(* IEC 61131-3 sources: volt/packages/volt-lsp-iec/test-corpus/lenze-mid/Device/Plc Logic/Application/Library Manager/RecipeManagement, 99 files *)

(* ---- IEC_ANYTYPE.dut ---- *)
TYPE IEC_ANYTYPE :
STRUCT
	PDATA : POINTER TO BYTE;
	TYPEOF : IEC_DataType;
	SIZE : UINT;
END_STRUCT
END_TYPE

(* ---- IEC_DATATYPE.dut ---- *)
TYPE IEC_DATATYPE :
(
	TYPE_BOOL,
	TYPE_INT,
	TYPE_BYTE,
	TYPE_WORD,
	TYPE_DINT,
	TYPE_DWORD,
	TYPE_REAL,
	TYPE_TIME,
	TYPE_STRING,
	TYPE_SINT,
	TYPE_USINT,
	TYPE_UINT,
	TYPE_UDINT,
	TYPE_DATE,
	TYPE_TOD,
	TYPE_DT,
	TYPE_LREAL,
	TYPE_LINT,
	TYPE_ULINT,
	TYPE_LWORD,
	TYPE_NONE,
	TYPE_BIT,
	TYPE_WSTRING,
	TYPE_LDATE,
	TYPE_LTOD,
	TYPE_LDT,
	TYPE_LTIME,
	TYPE_MAXTYPES
);
END_TYPE

(* ---- INFOVALUES.dut ---- *)
TYPE INFOVALUES :
(
	NO_INFO := 16#0,
	INFO_RECIPE_MANAGER_NOT_ALL_VARIABLES_FOUND := 16#1,
	INFO_RECIPE_MANAGER_OTHER_VARIABLES_FOUND := 16#2,
	INFO_RECIPE_MANAGER_ONE_OR_MORE_VARIABLES_FOUND := 16#4,
	INFO_RECIPE_MANAGER_ALL_VARIABLES_FOUND := 16#8
);
END_TYPE

(* ---- MEMBERSTOREDUCESTACKSIZE.dut ---- *)
TYPE MEMBERSTOREDUCESTACKSIZE :
STRUCT
	STFILE : STRING(512);
	TOKENIZER : RecipeManTokenizer;
	STPATHSEPARATOR : STRING(2);
	STHELP : STRING(512);
	STHELPPREVDIR : STRING(512);
	STCURRENTDIR : STRING(512);
	STLINEHELP : STRING(256);
	WSTVALUE : WSTRING(128);
	STHELPVALUE : STRING(256);
	STNAME : STRING(256);
	STRHELP : STRING(256);
END_STRUCT
END_TYPE

(* ---- MESSAGEBOX_STRUCT.dut ---- *)
TYPE MESSAGEBOX_STRUCT :
STRUCT
	EMESSAGEBOXDIALOGTYPES : DWORD;
	STITLE : STRING;
	SMESSAGETXT : STRING(1024);
END_STRUCT
END_TYPE

(* ---- PERSISTANTLOADTYPE.dut ---- *)
TYPE PERSISTANTLOADTYPE :
(
	LOAD_TYPE_NONE,
	LOAD_TYPE_SEARCH_FOR_NAME,
	LOAD_TYPE_SEARCH_FOR_VARNAME,
	LOAD_MATCHING_VARIABLES_BY_VARIABLENAME
);
END_TYPE

(* ---- RECIPEDATA.dut ---- *)
TYPE RECIPEDATA :
STRUCT
	PDATA : POINTER TO ARRAY [0..100000] OF RecipeDataValue;
	IDATACOUNT : DINT;
END_STRUCT
END_TYPE

(* ---- RECIPEDATAVALUE.dut ---- *)
TYPE RECIPEDATAVALUE :
STRUCT
	VALUE : IEC_AnyType;
END_STRUCT
END_TYPE

(* ---- RECIPEDESCRIPTION.dut ---- *)
TYPE RECIPEDESCRIPTION :
STRUCT
	STNAME : STRING;
	DATA : RecipeData;
	DESCDATA : RecipeDescriptionData;
END_STRUCT
END_TYPE

(* ---- RECIPEDESCRIPTIONDATA.dut ---- *)
TYPE RECIPEDESCRIPTIONDATA :
STRUCT
	PDATA : POINTER TO ARRAY [0..100000] OF RecipeVariableDescription;
	ICOUNT : DINT;
END_STRUCT
END_TYPE

(* ---- RECIPEMANENUMCOLUMNS.dut ---- *)
TYPE RECIPEMANENUMCOLUMNS :
(
	C_VARNAME,
	C_VALUE,
	C_TYPE,
	C_NAME,
	C_COMMENT,
	C_MIN,
	C_MAX
);
END_TYPE

(* ---- RECIPEREMOTEVARIABLE.dut ---- *)
TYPE RECIPEREMOTEVARIABLE :
STRUCT
	PBTINSTANCEPATH : POINTER TO BYTE;
END_STRUCT
END_TYPE

(* ---- RECIPEREMOTEVARIABLES.dut ---- *)
TYPE RECIPEREMOTEVARIABLES :
STRUCT
	PVARIABLES : POINTER TO RecipeRemoteVariable;
	DICOUNT : DINT;
END_STRUCT
END_TYPE

(* ---- RECIPESTORE.dut ---- *)
TYPE RECIPESTORE :
STRUCT
	_STPATH : STRING(512) := '';
	_BAUTOSAVE : BOOL := TRUE;
END_STRUCT
END_TYPE

(* ---- RECIPEVARIABLEDESCRIPTION.dut ---- *)
TYPE RECIPEVARIABLEDESCRIPTION :
STRUCT
	PSTNAME : POINTER TO BYTE;
	TYPEOF : IEC_DataType;
	MINVALUE : IEC_AnyType;
	MAXVALUE : IEC_AnyType;
	PSTVARNAME : POINTER TO BYTE;
	PSTCOMMENT : POINTER TO BYTE;
	DWFLAGS : DWORD;
END_STRUCT
END_TYPE

(* ---- STRINGINTPAIR.dut ---- *)
TYPE STRINGINTPAIR :
STRUCT
	STVAL : STRING(40);
	IVAL : INT;
END_STRUCT
END_TYPE

(* ---- GVL_RECIPECONSTANTS.gvl ---- *)
VAR_GLOBAL
	INVALID_DEFINITION_INDEX : INT := -1;
	CANNOT_ADD_RECIPE : INT := -1;
	INVALID_RECIPE_INDEX : INT := -1;
	RECIPESTORE_STRLEN : INT := 40;
	OUTPUT_INFO : INT := 16#1;
	OUTPUT_WARNING : INT := 16#2;
	OUTPUT_ERROR : INT := 16#4;
	OUTPUT_DEBUG : INT := 16#10;
	ASCII_PIPE : BYTE := 16#7C;
	NULL : POINTER TO BYTE := 0;
END_VAR

(* ---- GVL_RECIPEMANAGEMENT_INTERN.gvl ---- *)
VAR_GLOBAL
	G_RECIPEMANAGERCOMPONENT : STRING := 'RecipeManager';
	G_RECIPEMANAGERHELP : IRecipeManager;
	G_RECIPEMANCOMMANDSHELP : POINTER TO RecipeManCommands;
END_VAR

(* ---- GVL_RECIPEMANAGEMENT_TEMP.gvl ---- *)
VAR_GLOBAL
END_VAR

(* ---- GVL_RECIPEMANCOMMANDS_INTERN.gvl ---- *)
VAR_GLOBAL
	G_SEM : RecipeSem;
	G_BRECIPEMANAGERLOCKED : BOOL := TRUE;
	G_STFILENAME : STRING(512);
END_VAR

(* ---- INTERFACEIDS.gvl ---- *)
VAR_GLOBAL
	ITFID_IGENERIC : DWORD := 0;
	ITFID_IRECIPEMANAGER : DWORD := 1;
	ITFID_IGENERALCOMMAND : DWORD := 2;
END_VAR

(* ---- RETURNVALUES.gvl ---- *)
VAR_GLOBAL
	ERR_OK : UDINT := 16#0;
	ERR_FAILED : UDINT := 16#1;
	ERR_PARAMETER : UDINT := 16#2;
	ERR_NOTINITIALIZED : UDINT := 16#3;
	ERR_NOTIMPLEMENTED : UDINT := 16#C;
	ERR_NO_OBJECT : UDINT := 16#10;
	ERR_NOMEMORY : UDINT := 16#11;
	ERR_RECIPE_FILE_NOT_FOUND : UDINT := 16#4000;
	ERR_RECIPE_MISMATCH : UDINT := 16#4001;
	ERR_RECIPE_SAVE_ERR : UDINT := 16#4002;
	ERR_RECIPE_NOT_FOUND : UDINT := 16#4003;
	ERR_RECIPE_DEFINITION_NOT_FOUND : UDINT := 16#4004;
	ERR_RECIPE_ALREADY_EXIST : UDINT := 16#4005;
	ERR_NO_RECIPE_MANAGER_SET : UDINT := 16#4006;
	ERR_RECIPE_NOT_ALL_VARIABLES_WERE_LOADED : UDINT := 16#4007;
	ERR_RECIPE_NOMEMORY : UDINT := 16#4008;
	ERR_RECIPE_MANAGER_LOCKED_DURING_ONLINE_CHANGE : UDINT := 16#4009;
	ERR_SOURCE_EXHAUSTED : UDINT := 16#40A0;
	ERR_TARGET_EXHAUSTED : UDINT := 16#40A1;
	ERR_SOURCE_ILLEGAL : UDINT := 16#40A2;
END_VAR

(* ---- VERSIONINFO.gvl ---- *)
VAR_GLOBAL
	RECIPEMANAGER_VERSION_ATLEAST_3_2_0_0 : INT := 0;
	RECIPEMANAGER_VERSION_ATLEAST_3_2_0_1 : INT := 0;
	RECIPEMANAGER_VERSION_ATLEAST_3_2_0_2 : INT := 0;
	RECIPEMANAGER_VERSION_ATLEAST_3_3_0_0 : INT := 0;
	RECIPEMANAGER_VERSION_ATLEAST_3_3_0_10 : INT := 0;
	RECIPEMANAGER_VERSION_ATLEAST_3_3_0_20 : INT := 0;
	RECIPEMANAGER_VERSION_ATLEAST_3_5_5 : INT := 0;
	RECIPEMANAGER_VERSION_ATLEAST_3_5_9 : INT := 0;
	RECIPEMANAGER_VERSION_ATLEAST_3_5_10 : INT := 0;
	RECIPEMANAGER_VERSION_ATLEAST_3_5_14 : INT := 0;
END_VAR

(* ---- IGENERIC.itf ---- *)
INTERFACE IGENERIC
END_INTERFACE

METHOD GETINTERFACE : POINTER TO BYTE
VAR_INPUT
	DWITFID : DWORD;
END_VAR
END_METHOD

(* ---- IPERSISTANTRECIPELIST.itf ---- *)
INTERFACE IPERSISTANTRECIPELIST
END_INTERFACE

METHOD FREERECIPE : BOOL
VAR_INPUT
	RECIPE : IRecipe;
END_VAR
END_METHOD

METHOD GETRECIPENAME : STRING
VAR_INPUT
	IINDEX : INT;
END_VAR
END_METHOD

METHOD GETRECIPENAMES : DWORD
VAR_INPUT
	PSTRINGS : POINTER TO ARRAY [0..0] OF STRING;
	ISIZE : INT;
	ISTARTINDEX : INT;
END_VAR
END_METHOD

METHOD RELOAD : DWORD
END_METHOD

(* ---- IPERSISTANTRECIPELISTSUPPORTSADD.itf ---- *)
INTERFACE IPERSISTANTRECIPELISTSUPPORTSADD
END_INTERFACE

METHOD ADDRECIPE : BOOL
VAR_INPUT
	STNAME : REFERENCE TO STRING;
END_VAR
END_METHOD

(* ---- IPERSISTENTRECIPEHELPER.itf ---- *)
INTERFACE IPERSISTENTRECIPEHELPER
END_INTERFACE

METHOD DELETERECIPE : BOOL
VAR_INPUT
	STNAME : STRING;
END_VAR
END_METHOD

METHOD GETFILEEXTENSION : STRING
END_METHOD

METHOD GETFILEPATH : STRING(512)
END_METHOD

METHOD LOADRECIPE : BOOL
VAR_INPUT
	DESC : REFERENCE TO RecipeDescription;
END_VAR
END_METHOD

METHOD LOADRECIPEFROM : BOOL
VAR_INPUT
	DESC : REFERENCE TO RecipeDescription;
	STFILE : REFERENCE TO STRING(255);
END_VAR
END_METHOD

METHOD SAVERECIPE : BOOL
VAR_INPUT
	DESC : REFERENCE TO RecipeDescription;
END_VAR
END_METHOD

METHOD SAVERECIPEAS : BOOL
VAR_INPUT
	DESC : REFERENCE TO RecipeDescription;
	STFILE : REFERENCE TO STRING(255);
END_VAR
END_METHOD

METHOD SETFILEPATH : BOOL
VAR_INPUT
	STPATH : STRING(512);
END_VAR
END_METHOD

(* ---- IRECIPE.itf ---- *)
INTERFACE IRECIPE
END_INTERFACE

METHOD FILLDESCRIPTION : BOOL
VAR_INPUT
	DESC : REFERENCE TO RecipeDescription;
END_VAR
END_METHOD

METHOD READ : BOOL
END_METHOD

METHOD UPDATEFROMDESCRIPTION : BOOL
VAR_INPUT
	DESC : REFERENCE TO RecipeDescription;
END_VAR
END_METHOD

METHOD WRITE : BOOL
END_METHOD

(* ---- IRECIPECHECKONSTART.itf ---- *)
INTERFACE IRECIPECHECKONSTART
END_INTERFACE

METHOD ALREADYEXISTING : BOOL
VAR_INPUT
	STNAME : STRING;
END_VAR
END_METHOD

METHOD GETALREADYEXISTINGRECIPES : BOOL
END_METHOD

(* ---- IRECIPEDEFINITION.itf ---- *)
INTERFACE IRECIPEDEFINITION
END_INTERFACE

METHOD CREATERECIPE : BOOL
VAR_INPUT
	STNAME : STRING;
	BREADCURRENT : BOOL;
	BSAVE : BOOL;
END_VAR
END_METHOD

METHOD FREERECIPE : BOOL
VAR_INPUT
	RECIPE : IRecipe;
END_VAR
END_METHOD

METHOD GETPERSISTENCYHELPER : POINTER TO IPersistentRecipeHelper
END_METHOD

METHOD GETRECIPE : RecipeDescription
VAR_INPUT
	IINDEX : INT;
END_VAR
END_METHOD

METHOD GETRECIPEINDEXBYNAME : INT
VAR_INPUT
	STNAME : STRING;
END_VAR
END_METHOD

METHOD GETRECIPENAME : STRING
VAR_INPUT
	IINDEX : INT;
END_VAR
END_METHOD

METHOD GETRECIPENAMES : DWORD
VAR_INPUT
	PSTRINGS : POINTER TO ARRAY [0..0] OF STRING;
	ISIZE : INT;
	ISTARTINDEX : INT;
END_VAR
END_METHOD

METHOD GETRECIPEVALUES : DWORD
VAR_INPUT
	PSTRINGS : POINTER TO ARRAY [0..0] OF STRING;
	ISIZE : INT;
	ISTARTINDEX : INT;
	ISTRINGLENGTH : INT;
END_VAR
END_METHOD

METHOD GETRECIPEVARIABLENAMES : DWORD
VAR_INPUT
	PSTRINGS : POINTER TO ARRAY [0..0] OF STRING;
	ISIZE : INT;
	ISTARTINDEX : INT;
END_VAR
END_METHOD

METHOD LOADALL : BOOL
VAR_INPUT
	BCLEAR : BOOL;
END_VAR
END_METHOD

METHOD REGISTEREVENTHANDLER : BOOL
VAR_INPUT
	HANDLER : IRecipeDefinitionEventHandler;
END_VAR
END_METHOD

METHOD RELOAD : DWORD
END_METHOD

METHOD SAVEALL : BOOL
END_METHOD

METHOD SELECTRECIPE : BOOL
VAR_INPUT
	IINDEX : INT;
END_VAR
END_METHOD

METHOD SETRECIPEVALUES : DWORD
VAR_INPUT
	PSTRINGS : POINTER TO ARRAY [0..0] OF STRING;
	ISIZE : INT;
	ISTARTINDEX : INT;
END_VAR
END_METHOD

METHOD UNREGISTEREVENTHANDLER : BOOL
VAR_INPUT
	HANDLER : IRecipeDefinitionEventHandler;
END_VAR
END_METHOD

(* ---- IRECIPEDEFINITION2.itf ---- *)
INTERFACE IRECIPEDEFINITION2
END_INTERFACE

METHOD GETRECIPEVARIABLECOUNT : DINT
END_METHOD

METHOD GETRECIPEVARIABLENAME : POINTER TO BYTE
VAR_INPUT
	IVARINDEX : DINT;
END_VAR
VAR_OUTPUT
	ERRORCODE : DWORD;
END_VAR
END_METHOD

(* ---- IRECIPEDEFINITION3.itf ---- *)
INTERFACE IRECIPEDEFINITION3
END_INTERFACE

METHOD GETRECIPEVALUESSIZEOF : DWORD
VAR_INPUT
	PSTRINGS : POINTER TO ARRAY [0..0] OF STRING;
	ISIZE : INT;
	ISTARTINDEX : INT;
	ISIZEOFSTRING : INT;
END_VAR
END_METHOD

(* ---- IRECIPEDEFINITIONEVENTHANDLER.itf ---- *)
INTERFACE IRECIPEDEFINITIONEVENTHANDLER
END_INTERFACE

METHOD AFTERCREATE : BOOL
END_METHOD

METHOD BEFORECLEAR : BOOL
END_METHOD

METHOD SELECTIONCHANGED : BOOL
END_METHOD

(* ---- IRECIPEFACTORY.itf ---- *)
INTERFACE IRECIPEFACTORY
END_INTERFACE

METHOD CREATERECIPE : IRecipe
VAR_INPUT
	STDEFINITIONNAME : STRING;
	STRECIPENAME : STRING;
END_VAR
END_METHOD

METHOD FREERECIPE : BOOL
VAR_INPUT
	STDEFINITIONNAME : STRING;
	REC : IRecipe;
END_VAR
END_METHOD

(* ---- IRECIPEMANAGER.itf ---- *)
INTERFACE IRECIPEMANAGER
END_INTERFACE

METHOD GETRECIPEDEFINITION : IRecipeDefinition
VAR_INPUT
	IINDEX : INT;
END_VAR
END_METHOD

METHOD GETRECIPEDEFINITIONBYNAME : IRecipeDefinition
VAR_INPUT
	STDEFINITIONNAME : STRING;
END_VAR
END_METHOD

METHOD GETRECIPEDEFINITIONINDEXBYNAME : INT
VAR_INPUT
	STDEFINITIONNAME : STRING;
END_VAR
END_METHOD

METHOD SELECTRECIPEDEFINITION : BOOL
VAR_INPUT
	IINDEX : INT;
END_VAR
END_METHOD

(* ---- IRECIPESELECTION.itf ---- *)
INTERFACE IRECIPESELECTION
END_INTERFACE

METHOD DELETE : BOOL
END_METHOD

METHOD LOAD : BOOL
END_METHOD

METHOD LOADFROM : BOOL
VAR_INPUT
	STNAME : REFERENCE TO STRING(255);
END_VAR
END_METHOD

METHOD READ : BOOL
END_METHOD

METHOD READNOSAVE : BOOL
END_METHOD

METHOD RELEASE : BOOL
END_METHOD

METHOD SAVE : BOOL
END_METHOD

METHOD SAVEAS : BOOL
VAR_INPUT
	STNAME : REFERENCE TO STRING(255);
END_VAR
END_METHOD

METHOD UPDATEFROMVALUES : BOOL
VAR_INPUT
	DESC : RecipeDescription;
END_VAR
END_METHOD

METHOD WRITE : BOOL
END_METHOD

(* ---- IRECIPESELECTIONWITHCOMPARE.itf ---- *)
INTERFACE IRECIPESELECTIONWITHCOMPARE
END_INTERFACE

METHOD COMPARE : BOOL
END_METHOD

(* ---- IRECIPEWITHCOMPARE.itf ---- *)
INTERFACE IRECIPEWITHCOMPARE
END_INTERFACE

METHOD COMPARE : BOOL
END_METHOD

(* ---- ASSERT.pou ---- *)
FUNCTION ASSERT : BOOL
VAR_INPUT
	BVAL : BOOL;
	STMESSAGE : STRING;
END_VAR
END_FUNCTION

(* ---- DOFORFBSAVEASRECIPE.pou ---- *)
FUNCTION DOFORFBSAVEASRECIPE : BOOL
VAR_INPUT
	MEMORYFORFBSAVEASRECIPE : POINTER TO BYTE;
	RECIPEMAN : IRecipeManager;
	COMMANDMANAGER : ICommandManager2;
	ICMD : INT;
END_VAR
END_FUNCTION

(* ---- PSTRCAT.pou ---- *)
FUNCTION PSTRCAT : DINT
VAR_INPUT
	PSTDEST : POINTER TO STRING;
	PSTSRC : POINTER TO STRING;
	DIDESTSIZE : DINT;
END_VAR
END_FUNCTION

(* ---- PSTRLEN.pou ---- *)
FUNCTION PSTRLEN : DINT
VAR_INPUT
	PSTRING : POINTER TO STRING;
END_VAR
END_FUNCTION

(* ---- PSTRNCPY.pou ---- *)
FUNCTION PSTRNCPY : DINT
VAR_INPUT
	PSTDEST : POINTER TO BYTE;
	PSTSRC : POINTER TO BYTE;
	DIDESTSIZE : DINT;
END_VAR
END_FUNCTION

(* ---- RECIPEDODATASOURCESEXCHANGE.pou ---- *)
FUNCTION RECIPEDODATASOURCESEXCHANGE : UDINT
VAR_INPUT
	VARIABLES : RecipeRemoteVariables;
	BWRITING : BOOL;
	RECIPEMANAGER : IRecipeManager;
	DATASOURCESMGR : IDatasources.IDatasourcesMgr;
END_VAR
END_FUNCTION

(* ---- RECIPEDODATASOURCESEXCHANGE2.pou ---- *)
FUNCTION RECIPEDODATASOURCESEXCHANGE2 : UDINT
VAR_INPUT
	VARIABLES : RecipeRemoteVariables;
	RECIPEDEFNAME : STRING;
	BWRITING : BOOL;
	RECIPEMANAGER : IRecipeManager;
	DATASOURCESMGR : IDatasources.IDatasourcesMgr;
END_VAR
END_FUNCTION

(* ---- RECIPELOG.pou ---- *)
FUNCTION RECIPELOG : BOOL
VAR_INPUT
	DICLASS : DINT;
	DIERROR : DINT;
	DIINFO : DINT;
	STMESSAGE : STRING(255);
END_VAR
END_FUNCTION

(* ---- RECIPEMAN_FCTANYFROMSTRING.pou ---- *)
FUNCTION RECIPEMAN_FCTANYFROMSTRING : BOOL
VAR_INPUT
	STRSOURCE : POINTER TO STRING;
	PVARADR : POINTER TO BYTE;
	DWVARTYPE : IEC_DataType;
END_VAR
END_FUNCTION

(* ---- RECIPEMAN_FCTANYTOSTRING.pou ---- *)
FUNCTION RECIPEMAN_FCTANYTOSTRING : BOOL
VAR_INPUT
	STRRESULT : POINTER TO STRING;
	PVARADR : POINTER TO BYTE;
	DWVARTYPE : IEC_DataType;
END_VAR
END_FUNCTION

(* ---- RECIPEMAN_FCTDATATYPETOSTRING.pou ---- *)
FUNCTION RECIPEMAN_FCTDATATYPETOSTRING : BOOL
VAR_INPUT
	STRRESULT : POINTER TO STRING;
	DWVARTYPE : IEC_DataType;
END_VAR
END_FUNCTION

(* ---- RECIPEMAN_FCTGETDATAVALUE.pou ---- *)
FUNCTION RECIPEMAN_FCTGETDATAVALUE : POINTER TO BYTE
VAR_INPUT
	VALUE : IEC_AnyType;
	PSTR : POINTER TO BYTE;
	IBUFFERSIZE : INT;
	PILEN : POINTER TO INT;
END_VAR
END_FUNCTION

(* ---- RECIPEMAN_FCTLREALFROMSTRING.pou ---- *)
FUNCTION RECIPEMAN_FCTLREALFROMSTRING : BOOL
VAR_INPUT
	STRSOURCE : POINTER TO STRING;
	PVARADR : POINTER TO LREAL;
END_VAR
END_FUNCTION

(* ---- RECIPEMAN_FCTLREALTOSTRING.pou ---- *)
FUNCTION RECIPEMAN_FCTLREALTOSTRING : BOOL
VAR_INPUT
	STRRESULT : POINTER TO STRING;
	PVARADR : POINTER TO LREAL;
END_VAR
END_FUNCTION

(* ---- RECIPEMAN_FCTSETDATAVALUE.pou ---- *)
FUNCTION RECIPEMAN_FCTSETDATAVALUE : BOOL
VAR_INPUT
	DATA : POINTER TO BYTE;
	VALUE : IEC_AnyType;
END_VAR
END_FUNCTION

(* ---- RECIPEMAN_FCTSTRINGTODATATYPE.pou ---- *)
FUNCTION RECIPEMAN_FCTSTRINGTODATATYPE : BOOL
VAR_INPUT
	STRRESULT : POINTER TO STRING;
	DWVARTYPE : POINTER TO IEC_DataType;
END_VAR
END_FUNCTION

(* ---- RECIPEMAN_FCTTYPECLASSTODATATYPE.pou ---- *)
FUNCTION RECIPEMAN_FCTTYPECLASSTODATATYPE : IEC_DataType
VAR_INPUT
	TC : TypeClass;
END_VAR
END_FUNCTION

(* ---- RECIPEMAN_FILEEXISTS.pou ---- *)
FUNCTION RECIPEMAN_FILEEXISTS : BOOL
VAR_INPUT
	STFILENAME : REFERENCE TO STRING(255);
END_VAR
END_FUNCTION

(* ---- RECIPEMANCREATEDIRECTORY.pou ---- *)
FUNCTION RECIPEMANCREATEDIRECTORY : DWORD
VAR_INPUT
	PSTPATH : POINTER TO STRING(512);
	PMTRSS : POINTER TO MembersToReduceStackSize;
END_VAR
END_FUNCTION

(* ---- RECIPEMANMASKSTRING.pou ---- *)
FUNCTION RECIPEMANMASKSTRING : STRING(256)
VAR_INPUT
	PSTR : POINTER TO STRING(256);
	BWITHSEPARATOR : BOOL;
	CHSEPARATOR : BYTE;
	BFORUTF8 : BOOL;
END_VAR
END_FUNCTION

(* ---- RECIPEMANMASKWSTRING.pou ---- *)
FUNCTION RECIPEMANMASKWSTRING : BOOL
VAR_INPUT
	PBYTEIN : POINTER TO ARRAY [0..0] OF BYTE;
	PBYTEOUT : POINTER TO ARRAY [0..0] OF BYTE;
	IBUFFERSIZE : INT;
	BFORUTF8 : BOOL;
END_VAR
END_FUNCTION

(* ---- RECIPEMANUNMASKSTRING.pou ---- *)
FUNCTION RECIPEMANUNMASKSTRING : STRING(256)
VAR_INPUT
	PSTR : POINTER TO STRING(256);
	BWITHSEPARATOR : BOOL;
	CHSEPARATOR : BYTE;
	BFORUTF8 : BOOL;
END_VAR
END_FUNCTION

(* ---- RECIPEMANUNMASKWSTRING.pou ---- *)
FUNCTION RECIPEMANUNMASKWSTRING : BOOL
VAR_INPUT
	PSTR : POINTER TO STRING(256);
	BFORUTF8 : BOOL;
END_VAR
END_FUNCTION

(* ---- RECIPEMANWSTRINGTOSTRING.pou ---- *)
FUNCTION RECIPEMANWSTRINGTOSTRING : BOOL
VAR_INPUT
	PWSTRINGFROM : POINTER TO WSTRING;
	PSTRINGTO : POINTER TO STRING;
END_VAR
END_FUNCTION

(* ---- RECIPEPSTRNCPY.pou ---- *)
FUNCTION RECIPEPSTRNCPY : DINT
VAR_INPUT
	PSTDEST : POINTER TO BYTE;
	PSTSRC : POINTER TO BYTE;
	DIDESTSIZE : DINT;
END_VAR
END_FUNCTION

(* ---- RECIPESTRCMP.pou ---- *)
FUNCTION RECIPESTRCMP : INT
VAR_INPUT
	PST1 : POINTER TO STRING;
	PST2 : POINTER TO STRING;
	BENDSWITH : BOOL;
END_VAR
END_FUNCTION

(* ---- UTILGETFILESIZE.pou ---- *)
FUNCTION UTILGETFILESIZE : __XWORD
VAR_INPUT
	DWHANDLE : SysFile.RTS_IEC_HANDLE;
	STFILENAME : REFERENCE TO STRING(255);
	PULRESULT : POINTER TO UDINT;
END_VAR
END_FUNCTION

(* ---- VISU_FCTGETRECIPEDEFINITION.pou ---- *)
FUNCTION VISU_FCTGETRECIPEDEFINITION : DWORD
VAR_INPUT
	DWPARAM1 : __XWORD;
	DWPARAM2 : __XWORD;
	RECIPEMANAGER : IRecipeManager;
END_VAR
VAR_OUTPUT
	_RECIPEDEFINITION : IRecipeDefinition;
END_VAR
END_FUNCTION

(* ---- VISU_FCTGETRECIPEDEFINITION2.pou ---- *)
FUNCTION VISU_FCTGETRECIPEDEFINITION2 : DWORD
VAR_INPUT
	DWPARAM1 : __XWORD;
	DWPARAM2 : __XWORD;
	RECIPEMANAGER : IRecipeManager;
	BNOCURRENTRECIPEDEFINITION : BOOL;
END_VAR
VAR_OUTPUT
	_RECIPEDEFINITION : IRecipeDefinition;
END_VAR
END_FUNCTION

(* ---- VISU_FCTGETRECIPESELECTION.pou ---- *)
FUNCTION VISU_FCTGETRECIPESELECTION : DWORD
VAR_INPUT
	DWPARAM1 : __XWORD;
	DWPARAM2 : __XWORD;
	RECIPEMANAGER : IRecipeManager;
END_VAR
VAR_OUTPUT
	_RECIPEDEFINITION : IRecipeDefinition;
	_RECIPESELECTION : IRecipeSelection;
END_VAR
END_FUNCTION

(* ---- VISU_FCTGETRECIPESELECTION2.pou ---- *)
FUNCTION VISU_FCTGETRECIPESELECTION2 : DWORD
VAR_INPUT
	DWPARAM1 : __XWORD;
	DWPARAM2 : __XWORD;
	RECIPEMANAGER : IRecipeManager;
	BNOCURRENTRECIPESELECTION : BOOL;
END_VAR
VAR_OUTPUT
	_RECIPEDEFINITION : IRecipeDefinition;
	_RECIPESELECTION : IRecipeSelection;
END_VAR
END_FUNCTION

(* ---- ABSTRACTFILEPARAMSCOMMAND.pou ---- *)
FUNCTION_BLOCK ABSTRACTFILEPARAMSCOMMAND EXTENDS AbstractGeneralCommand
END_FUNCTION_BLOCK

METHOD EXECUTE : __XWORD
VAR_INPUT
	DWPARAM1 : __XWORD;
	DWPARAM2 : __XWORD;
END_VAR
END_METHOD

METHOD EXECUTEONFILEPARAMS : DWORD
VAR_INPUT
	STRECIPEDEF : STRING;
	STRECIPENAME : STRING;
	STFILE : STRING(255);
END_VAR
END_METHOD

(* ---- ABSTRACTGENERALCOMMAND.pou ---- *)
FUNCTION_BLOCK ABSTRACTGENERALCOMMAND
VAR
	_ITFGENERALCOMMAND : IGeneralCommand2 := THIS^;
	_RECIPEMANAGER : IRecipeManager;
	S_BASECOMMANDS : RecipeManCommands;
END_VAR
END_FUNCTION_BLOCK

METHOD EXECUTE : __XWORD
VAR_INPUT
	DWPARAM1 : __XWORD;
	DWPARAM2 : __XWORD;
END_VAR
END_METHOD

METHOD GETINTERFACE : POINTER TO BYTE
VAR_INPUT
	DWITFID : DWORD;
END_VAR
END_METHOD

METHOD SETRECIPEMANAGER
VAR_INPUT
	RECIPEMANAGER : IRecipeManager;
END_VAR
END_METHOD

(* ---- ABSTRACTRECIPEANDDEFINITIONNAMECOMMAND.pou ---- *)
FUNCTION_BLOCK ABSTRACTRECIPEANDDEFINITIONNAMECOMMAND EXTENDS AbstractGeneralCommand
END_FUNCTION_BLOCK

METHOD EXECUTE : __XWORD
VAR_INPUT
	DWPARAM1 : __XWORD;
	DWPARAM2 : __XWORD;
END_VAR
END_METHOD

METHOD EXECUTEONRECIPEDEFINITIONANDRECIPENAME : DWORD
VAR_INPUT
	STRECIPEDEFINITIONNAME : STRING;
	STRECIPENAME : STRING;
END_VAR
END_METHOD

(* ---- BINARYMANYFILESPERSISTANTRECIPEHELPER.pou ---- *)
FUNCTION_BLOCK BINARYMANYFILESPERSISTANTRECIPEHELPER
VAR
	_STDEFNAME : STRING;
	_STEXTENSION : STRING(16) := '.binrecipe';
	_STPATH : STRING(512) := '';
	_RECIPEMANAGER : IRecipeManager;
	_DATABUFFER : ARRAY [0..MAX_BUFFER_SIZE] OF BYTE;
	_CURRENTDATAPOSITION : INT;
	_MTRSS : MembersToReduceStackSize;
	MAX_BUFFER_SIZE : INT := 2000;
	RECIPEDEFINITIONNAME : STRING;
END_VAR
END_FUNCTION_BLOCK

METHOD DELETERECIPE : BOOL
VAR_INPUT
	STNAME : STRING;
END_VAR
END_METHOD

METHOD GETFILEEXTENSION : STRING
END_METHOD

METHOD GETFILEPATH : STRING(512)
END_METHOD

METHOD LOADRECIPE : BOOL
VAR_INPUT
	DESC : REFERENCE TO RecipeDescription;
END_VAR
END_METHOD

METHOD LOADRECIPEFROM : BOOL
VAR_INPUT
	DESC : REFERENCE TO RecipeDescription;
	STFILE : REFERENCE TO STRING(255);
END_VAR
END_METHOD

METHOD SAVERECIPE : BOOL
VAR_INPUT
	DESC : REFERENCE TO RecipeDescription;
END_VAR
END_METHOD

METHOD SAVERECIPEAS : BOOL
VAR_INPUT
	DESC : REFERENCE TO RecipeDescription;
	STFILE : REFERENCE TO STRING(255);
END_VAR
END_METHOD

METHOD SETFILEPATH : BOOL
VAR_INPUT
	STPATH : STRING(512);
END_VAR
END_METHOD

METHOD SETRECIPEMANAGER
VAR_INPUT
	RECIPEMANAGER : IRecipeManager;
END_VAR
END_METHOD

METHOD PRVINITFILENAME : BOOL
VAR_INPUT
	STRECIPE : STRING;
END_VAR
END_METHOD

METHOD PRVMEMCOPY : BOOL
VAR_INPUT
	PMEMDEST : POINTER TO BYTE;
	PMEMSOURCE : POINTER TO BYTE;
	ISIZE : INT;
END_VAR
END_METHOD

METHOD PRVREADDATAVALUE : BOOL
VAR_INPUT
	VALUE : IEC_AnyType;
	DWFILE : SysFile.RTS_IEC_HANDLE;
END_VAR
END_METHOD

METHOD PRVREADVALUE : BOOL
VAR_INPUT
	PDATA : POINTER TO BYTE;
	TYPEOF : IEC_DataType;
	VALUESIZE : UINT;
	DWFILE : SysFile.RTS_IEC_HANDLE;
END_VAR
END_METHOD

METHOD PRVSAVERECIPEBUFFERED : BOOL
VAR_INPUT
	DESC : REFERENCE TO RecipeDescription;
	DWHANDLE : SysFile.RTS_IEC_HANDLE;
END_VAR
END_METHOD

METHOD PRVSETLASTERROR : BOOL
VAR_INPUT
	DWERROR : DWORD;
END_VAR
END_METHOD

METHOD PRVWRITEDATAVALUE : BOOL
VAR_INPUT
	VALUE : IEC_AnyType;
	DWFILE : SysFile.RTS_IEC_HANDLE;
END_VAR
END_METHOD

METHOD PRVWRITEVALUE : BOOL
VAR_INPUT
	PDATA : POINTER TO BYTE;
	ISIZE : INT;
	TYPEOF : IEC_DataType;
	DWFILE : SysFile.RTS_IEC_HANDLE;
END_VAR
END_METHOD

METHOD PRVWRITEVALUEBUFFERED : BOOL
VAR_INPUT
	DWFILE : SysFile.RTS_IEC_HANDLE;
	PDATA : POINTER TO BYTE;
	ISIZE : INT;
END_VAR
END_METHOD

(* ---- PERSISTANTRECIPELIST.pou ---- *)
FUNCTION_BLOCK PERSISTANTRECIPELIST
VAR_INPUT
	_IPERSISTENTRECIPEHELPER : IPersistentRecipeHelper;
END_VAR
VAR
	_RECIPESVECTOR : Collections.StringVector;
	_TOKENIZER : RecipeManTokenizer;
	_STATICMEM : ARRAY [0..(STATIC_RECIPE_NAMES_SIZE / 4)] OF DWORD;
	STATIC_RECIPE_NAMES_SIZE : DWORD := 2000;
	RECIPECOUNT : INT;
END_VAR
END_FUNCTION_BLOCK

METHOD ADDRECIPE : BOOL
VAR_INPUT
	STNAME : REFERENCE TO STRING;
END_VAR
END_METHOD

METHOD FB_EXIT : BOOL
VAR_INPUT
	BINCOPYCODE : BOOL;
END_VAR
END_METHOD

METHOD FB_INIT : BOOL
VAR_INPUT
	BINITRETAINS : BOOL;
	BINCOPYCODE : BOOL;
END_VAR
END_METHOD

METHOD FREERECIPE : BOOL
VAR_INPUT
	RECIPE : IRecipe;
END_VAR
END_METHOD

METHOD GETRECIPENAME : STRING
VAR_INPUT
	IINDEX : INT;
END_VAR
END_METHOD

METHOD GETRECIPENAMES : DWORD
VAR_INPUT
	PSTRINGS : POINTER TO ARRAY [0..0] OF STRING;
	ISIZE : INT;
	ISTARTINDEX : INT;
END_VAR
END_METHOD

METHOD RELOAD : DWORD
END_METHOD

METHOD PRVADD : BOOL
VAR_INPUT
	STRECIPEFILE : REFERENCE TO STRING;
END_VAR
END_METHOD

METHOD PRVCLEAR : BOOL
END_METHOD

(* ---- RECIPECOLLECTION.pou ---- *)
FUNCTION_BLOCK RECIPECOLLECTION
VAR
	_ASTATICRECIPES : ARRAY [0..STATIC_RECIPE_COUNT] OF IRecipe;
	_IUSEDRECIPES : INT;
	_PADYNAMICRECIPES : POINTER TO ARRAY [0..20] OF IRecipe := 0;
	_IDYNAMICALLOCCOUNT : INT;
	STATIC_RECIPE_COUNT : INT := 20;
	FIRST_DYNAMIC_ALLOC_COUNT : INT := 20;
	COUNT : INT;
END_VAR
END_FUNCTION_BLOCK

METHOD ADDRECIPE : BOOL
VAR_INPUT
	RECIPE : IRecipe;
END_VAR
END_METHOD

METHOD FB_EXIT : BOOL
VAR_INPUT
	BINCOPYCODE : BOOL;
END_VAR
END_METHOD

METHOD GETRECIPE : IRecipe
VAR_INPUT
	IINDEX : INT;
END_VAR
END_METHOD

METHOD GETRECIPENAMES : DWORD
VAR_INPUT
	PSTRINGS : POINTER TO ARRAY [0..0] OF STRING;
	ISIZE : INT;
	ISTARTINDEX : INT;
END_VAR
END_METHOD

METHOD REMOVERECIPE : BOOL
VAR_INPUT
	IINDEX : INT;
END_VAR
END_METHOD

(* ---- RECIPEDEFINITION.pou ---- *)
FUNCTION_BLOCK RECIPEDEFINITION
VAR
	_STNAME : STRING;
	_PERSISTANTRECIPELIST : PersistantRecipeList;
	_IRECIPELIST : IPersistantRecipeList;
	_ICURRENTRECIPE : IRecipe := 0;
	_RECIPECOLL : RecipeCollection;
	_EVENTHELPER : RecipeDefinitionEventHelper;
	_PPERSISTENCYHELPER : POINTER TO IPersistentRecipeHelper;
	_BAUTOSAVE : BOOL := TRUE;
	_RECDESC : RecipeDescription;
	_CURSOR : RecipeSelection;
	_ICURRENTINDEX : INT := -1;
	_IRETURNEDINDEX : INT := -1;
	_INTERNALRECDESC : RecipeDescription;
	_RECIPEMANAGER : IRecipeManager;
	_RECIPEFACTORY : IRecipeFactory;
	ARRALREADYEXISTINGFILES : POINTER TO ARRAY [0..0] OF STRING(80);
	_IALREADYEXISTINGRECIPES : INT;
	CURRENT : IRecipeSelection;
	CURRENTLYSELECTEDRECIPE : POINTER TO RecipeDescription;
	INTPERSISTENCY : BOOL;
	NAME : STRING;
	PRVCURRENTRECIPE : IRecipe;
	PRVRECIPELIST : IPersistantRecipeList;
	RECIPECOUNT : INT;
END_VAR
END_FUNCTION_BLOCK

METHOD ALREADYEXISTING : BOOL
VAR_INPUT
	STNAME : STRING;
END_VAR
END_METHOD

METHOD CREATERECIPE : BOOL
VAR_INPUT
	STNAME : STRING;
	BREADCURRENT : BOOL;
	BSAVE : BOOL;
END_VAR
END_METHOD

METHOD FB_EXIT : BOOL
VAR_INPUT
	BINCOPYCODE : BOOL;
END_VAR
END_METHOD

METHOD FREERECIPE : BOOL
VAR_INPUT
	RECIPE : IRecipe;
END_VAR
END_METHOD

METHOD GETALREADYEXISTINGRECIPES : BOOL
END_METHOD

METHOD GETPERSISTENCYHELPER : POINTER TO IPersistentRecipeHelper
END_METHOD

METHOD GETRECIPE : RecipeDescription
VAR_INPUT
	IINDEX : INT;
END_VAR
END_METHOD

METHOD GETRECIPEBYNAME : IRecipe
VAR_INPUT
	STNAME : REFERENCE TO STRING;
END_VAR
END_METHOD

METHOD GETRECIPEINDEXBYNAME : INT
VAR_INPUT
	STNAME : STRING;
END_VAR
END_METHOD

METHOD GETRECIPENAME : STRING
VAR_INPUT
	IINDEX : INT;
END_VAR
END_METHOD

METHOD GETRECIPENAMES : DWORD
VAR_INPUT
	PSTRINGS : POINTER TO ARRAY [0..0] OF STRING;
	ISIZE : INT;
	ISTARTINDEX : INT;
END_VAR
END_METHOD

METHOD GETRECIPEVALUES : DWORD
VAR_INPUT
	PSTRINGS : POINTER TO ARRAY [0..0] OF STRING;
	ISIZE : INT;
	ISTARTINDEX : INT;
	ISTRINGLENGTH : INT;
END_VAR
END_METHOD

METHOD GETRECIPEVALUESSIZEOF : DWORD
VAR_INPUT
	PSTRINGS : POINTER TO ARRAY [0..0] OF STRING;
	ISIZE : INT;
	ISTARTINDEX : INT;
	ISIZEOFSTRING : INT;
END_VAR
END_METHOD

METHOD GETRECIPEVARIABLECOUNT : DINT
END_METHOD

METHOD GETRECIPEVARIABLENAME : POINTER TO BYTE
VAR_INPUT
	IVARINDEX : DINT;
END_VAR
VAR_OUTPUT
	ERRORCODE : DWORD;
END_VAR
END_METHOD

METHOD GETRECIPEVARIABLENAMES : DWORD
VAR_INPUT
	PSTRINGS : POINTER TO ARRAY [0..0] OF STRING;
	ISIZE : INT;
	ISTARTINDEX : INT;
END_VAR
END_METHOD

METHOD LOADALL : BOOL
VAR_INPUT
	BCLEAR : BOOL;
END_VAR
END_METHOD

METHOD REGISTEREVENTHANDLER : BOOL
VAR_INPUT
	HANDLER : IRecipeDefinitionEventHandler;
END_VAR
END_METHOD

METHOD RELOAD : DWORD
END_METHOD

METHOD SAVEALL : BOOL
END_METHOD

METHOD SELECTRECIPE : BOOL
VAR_INPUT
	IINDEX : INT;
END_VAR
END_METHOD

METHOD SETRECIPEFACTORY
VAR_INPUT
	RECIPEFACTORY : IRecipeFactory;
END_VAR
END_METHOD

METHOD SETRECIPEMANAGER
VAR_INPUT
	RECIPEMANAGER : IRecipeManager;
END_VAR
END_METHOD

METHOD SETRECIPEVALUES : DWORD
VAR_INPUT
	PSTRINGS : POINTER TO ARRAY [0..0] OF STRING;
	ISIZE : INT;
	ISTARTINDEX : INT;
END_VAR
END_METHOD

METHOD UNREGISTEREVENTHANDLER : BOOL
VAR_INPUT
	HANDLER : IRecipeDefinitionEventHandler;
END_VAR
END_METHOD

METHOD INTGETINTERNALRECIPEDESCRIPTION : POINTER TO RecipeDescription
END_METHOD

METHOD PRVAUTOSAVE : BOOL
END_METHOD

METHOD PRVCLEAR : BOOL
END_METHOD

METHOD PRVGETVALUE : BOOL
VAR_INPUT
	VALUE : IEC_AnyType;
	PSTR : POINTER TO BYTE;
	IBUFFERSIZE : INT;
	PILEN : POINTER TO INT;
END_VAR
END_METHOD

METHOD PRVSETVALUE : BOOL
VAR_INPUT
	DATA : POINTER TO BYTE;
	VALUE : IEC_AnyType;
END_VAR
END_METHOD

(* ---- RECIPEDEFINITIONEVENTHELPER.pou ---- *)
FUNCTION_BLOCK RECIPEDEFINITIONEVENTHELPER
VAR
	_HANDLERS : ARRAY [0..MAXNUM] OF IRecipeDefinitionEventHandler;
	_IREGISTEREDHANDLERCOUNT : INT;
	MAXNUM : INT := 3;
END_VAR
END_FUNCTION_BLOCK

METHOD AFTERCREATE : BOOL
END_METHOD

METHOD BEFORECLEAR : BOOL
END_METHOD

METHOD REGISTER : BOOL
VAR_INPUT
	HANDLER : IRecipeDefinitionEventHandler;
END_VAR
END_METHOD

METHOD SELECTIONCHANGED : BOOL
END_METHOD

METHOD UNREGISTER : BOOL
VAR_INPUT
	HANDLER : IRecipeDefinitionEventHandler;
END_VAR
END_METHOD

(* ---- RECIPEMANAGER.pou ---- *)
FUNCTION_BLOCK RECIPEMANAGER
VAR
	_ARRDEFINITIONS : POINTER TO ARRAY [0..1000] OF IRecipeDefinition;
	_IDEFINITIONCOUNT : INT;
	_INEXTTOINSERTINDEX : INT;
	_ICURRENTINDEX : INT := -1;
	_IRECIPEMANAGER : IRecipeManager;
	_UDILASTERROR : UDINT;
	_ELASTINFO : InfoValues;
	CURRENT : IRecipeDefinition;
	DEFINITIONCOUNT : INT;
	LASTERROR : UDINT;
	LASTINFO : InfoValues;
END_VAR
END_FUNCTION_BLOCK

METHOD ADDRECIPEDEFINITION : BOOL
VAR_INPUT
	DEF : IRecipeDefinition;
END_VAR
END_METHOD

METHOD FB_INIT : BOOL
VAR_INPUT
	BINITRETAINS : BOOL;
	BINCOPYCODE : BOOL;
END_VAR
END_METHOD

METHOD GETINTERFACE : POINTER TO BYTE
VAR_INPUT
	DWITFID : DWORD;
END_VAR
END_METHOD

METHOD GETRECIPEDEFINITION : IRecipeDefinition
VAR_INPUT
	IINDEX : INT;
END_VAR
END_METHOD

METHOD GETRECIPEDEFINITIONBYNAME : IRecipeDefinition
VAR_INPUT
	STDEFINITIONNAME : STRING;
END_VAR
END_METHOD

METHOD GETRECIPEDEFINITIONINDEXBYNAME : INT
VAR_INPUT
	STDEFINITIONNAME : STRING;
END_VAR
END_METHOD

METHOD INITIALIZE : BOOL
VAR_INPUT
	PDATA : POINTER TO ARRAY [0..1000] OF IRecipeDefinition;
	ICOUNT : INT;
END_VAR
END_METHOD

METHOD SELECTRECIPEDEFINITION : BOOL
VAR_INPUT
	IINDEX : INT;
END_VAR
END_METHOD

(* ---- RECIPEMANCOMMANDS.pou ---- *)
FUNCTION_BLOCK RECIPEMANCOMMANDS
VAR
	_RECIPEMANAGER : IRecipeManager;
	_RECIPEDEFINITION : IRecipeDefinition;
	_BRECIPEMANAGERSET : BOOL;
END_VAR
END_FUNCTION_BLOCK

METHOD CREATERECIPE : DWORD
VAR_IN_OUT
	RECIPEDEFINITIONNAME : STRING;
	RECIPENAME : STRING;
END_VAR
END_METHOD

METHOD CREATERECIPENOSAVE : DWORD
VAR_IN_OUT
	RECIPEDEFINITIONNAME : STRING;
	RECIPENAME : STRING;
END_VAR
END_METHOD

METHOD DELETERECIPE : DWORD
VAR_IN_OUT
	RECIPEDEFINITIONNAME : STRING;
	RECIPENAME : STRING;
END_VAR
END_METHOD

METHOD DELETERECIPEFILE : DWORD
VAR_IN_OUT
	RECIPEDEFINITIONNAME : STRING;
	RECIPENAME : STRING;
END_VAR
END_METHOD

METHOD GETLASTERROR : DWORD
END_METHOD

METHOD GETLASTINFO : InfoValues
END_METHOD

METHOD GETRECIPECOUNT : INT
VAR_IN_OUT
	RECIPEDEFINITIONNAME : STRING;
END_VAR
END_METHOD

METHOD GETRECIPENAMES : DWORD
VAR_INPUT
	PSTRINGS : POINTER TO ARRAY [0..0] OF STRING;
	ISIZE : INT;
	ISTARTINDEX : INT;
END_VAR
VAR_IN_OUT
	RECIPEDEFINITIONNAME : STRING;
END_VAR
END_METHOD

METHOD GETRECIPEVALUES : DWORD
VAR_INPUT
	PSTRINGS : POINTER TO ARRAY [0..0] OF STRING;
	ISIZE : INT;
	ISTARTINDEX : INT;
	ISTRINGLENGTH : INT;
END_VAR
VAR_IN_OUT
	RECIPEDEFINITIONNAME : STRING;
	RECIPENAME : STRING;
END_VAR
END_METHOD

METHOD GETRECIPEVALUESSIZEOF : DWORD
VAR_INPUT
	PSTRINGS : POINTER TO ARRAY [0..0] OF STRING;
	ISIZE : INT;
	ISTARTINDEX : INT;
	ISIZEOFSTRING : INT;
END_VAR
VAR_IN_OUT
	RECIPEDEFINITIONNAME : STRING;
	RECIPENAME : STRING;
END_VAR
END_METHOD

METHOD GETRECIPEVARIABLENAMES : DWORD
VAR_INPUT
	PSTRINGS : POINTER TO ARRAY [0..0] OF STRING;
	ISIZE : INT;
	ISTARTINDEX : INT;
END_VAR
VAR_IN_OUT
	RECIPEDEFINITIONNAME : STRING;
	RECIPENAME : STRING;
END_VAR
END_METHOD

METHOD LOADANDWRITERECIPE : DWORD
VAR_IN_OUT
	RECIPEDEFINITIONNAME : STRING;
	RECIPENAME : STRING;
END_VAR
END_METHOD

METHOD LOADFROMANDWRITERECIPE : DWORD
VAR_IN_OUT
	RECIPEDEFINITIONNAME : STRING;
	RECIPENAME : STRING;
	FILENAME : STRING(255);
END_VAR
END_METHOD

METHOD LOADRECIPE : DWORD
VAR_IN_OUT
	RECIPEDEFINITIONNAME : STRING;
	RECIPENAME : STRING;
END_VAR
END_METHOD

METHOD READANDSAVEAS : DWORD
VAR_IN_OUT
	RECIPEDEFINITIONNAME : STRING;
	FILENAME : STRING(255);
END_VAR
END_METHOD

METHOD READANDSAVERECIPE : DWORD
VAR_IN_OUT
	RECIPEDEFINITIONNAME : STRING;
	RECIPENAME : STRING;
END_VAR
END_METHOD

METHOD READANDSAVERECIPEAS : DWORD
VAR_IN_OUT
	RECIPEDEFINITIONNAME : STRING;
	RECIPENAME : STRING;
	FILENAME : STRING(255);
END_VAR
END_METHOD

METHOD READRECIPE : DWORD
VAR_IN_OUT
	RECIPEDEFINITIONNAME : STRING;
	RECIPENAME : STRING;
END_VAR
END_METHOD

METHOD REGISTERDATASOURCERECIPEDEFINITION : DWORD
VAR_INPUT
	DATASOURCESMGR : IDatasources.IDatasourcesMgr;
END_VAR
VAR_IN_OUT
	RECIPEDEFINITIONNAME : STRING;
END_VAR
END_METHOD

METHOD RELOADRECIPES : DWORD
VAR_IN_OUT
	RECIPEDEFINITIONNAME : STRING;
END_VAR
END_METHOD

METHOD RESETLASTERROR : DWORD
END_METHOD

METHOD RESETLASTINFO : DWORD
END_METHOD

METHOD SAVERECIPE : DWORD
VAR_IN_OUT
	RECIPEDEFINITIONNAME : STRING;
	RECIPENAME : STRING;
END_VAR
END_METHOD

METHOD SETRECIPEVALUES : DWORD
VAR_INPUT
	PSTRINGS : POINTER TO ARRAY [0..0] OF STRING;
	ISIZE : INT;
	ISTARTINDEX : INT;
END_VAR
VAR_IN_OUT
	RECIPEDEFINITIONNAME : STRING;
	RECIPENAME : STRING;
END_VAR
END_METHOD

METHOD SETSTORAGEPATH : BOOL
VAR_INPUT
	STPATH : STRING(512);
END_VAR
END_METHOD

METHOD WRITERECIPE : DWORD
VAR_IN_OUT
	RECIPEDEFINITIONNAME : STRING;
	RECIPENAME : STRING;
END_VAR
END_METHOD

METHOD SETRECIPEMANAGER : DWORD
VAR_INPUT
	RECIPEMANAGER : IRecipeManager;
END_VAR
END_METHOD

METHOD PRVCHECKRECIPEMANAGER : BOOL
VAR_INPUT
	BRESETLASTERROR : BOOL;
END_VAR
END_METHOD

METHOD PRVCOMPARERECIPE : BOOL
VAR_IN_OUT
	RECIPEDEFINITIONNAME : STRING;
	RECIPENAME : STRING;
END_VAR
END_METHOD

METHOD PRVCREATERECIPEHELP : DWORD
VAR_INPUT
	BSAVE : BOOL;
END_VAR
VAR_IN_OUT
	RECIPEDEFINITIONNAME : STRING;
	RECIPENAME : STRING;
END_VAR
END_METHOD

METHOD PRVGETRECIPEDEFINTIONBYNAME : IRecipeDefinition
VAR_IN_OUT
	STRECIPEDEF : STRING;
END_VAR
END_METHOD

METHOD PRVGETRECIPESELECTION : IRecipeSelection
VAR_IN_OUT
	STRECIPEDEF : STRING;
	STRECIPE : STRING;
END_VAR
END_METHOD

METHOD PRVREADANDSAVEAS : DWORD
VAR_IN_OUT
	RECIPEDEFINITIONNAME : STRING;
	FILENAME : STRING(255);
END_VAR
END_METHOD

METHOD PRVSETRECIPEDEFINITION : DWORD
VAR_IN_OUT
	RECIPEDEFINITIONNAME : STRING;
	RECIPENAME : STRING;
END_VAR
END_METHOD

(* ---- RECIPEMANTOKENIZER.pou ---- *)
FUNCTION_BLOCK RECIPEMANTOKENIZER
VAR
	_PSTRTOTOKENIZE : POINTER TO STRING;
	_PSTRTOTOKENIZEASBYTES : POINTER TO BYTE;
	_STRDELIMS : STRING(2);
	_INUMDELIMS : INT;
	_ICURRENTPOS : INT;
	_ISTRTOTOKENIZELEN : DINT;
	CURRENTPOSITION : INT;
END_VAR
END_FUNCTION_BLOCK

METHOD INITIALIZE : BOOL
VAR_INPUT
	PSTR : POINTER TO STRING;
	STRDELIMS : STRING;
END_VAR
END_METHOD

METHOD ISDELIMITER : BOOL
END_METHOD

METHOD NEXTLENGTHTOKEN : STRING(256)
VAR_INPUT
	NLENGTH : INT;
END_VAR
VAR_OUTPUT
	BEND : BOOL;
	ITOKENSTARTOFFSET : DINT;
	ITOKENENDOFFSET : DINT;
END_VAR
END_METHOD

METHOD NEXTSTRINGTOKEN : STRING(256)
VAR_INPUT
	PBEMPTYVALUE : POINTER TO BOOL;
END_VAR
VAR_OUTPUT
	BEND : BOOL;
	ITOKENSTARTOFFSET : DINT;
	ITOKENENDOFFSET : DINT;
END_VAR
END_METHOD

METHOD NEXTTOKEN : STRING(256)
VAR_OUTPUT
	BEND : BOOL;
	ITOKENSTARTOFFSET : DINT;
	ITOKENENDOFFSET : DINT;
END_VAR
END_METHOD

(* ---- RECIPESELECTION.pou ---- *)
FUNCTION_BLOCK RECIPESELECTION
VAR
	_RECIPE : IRecipe;
	_PRECIPEDEF : POINTER TO RecipeDefinition;
	_PPERSISTENCYHELPER : POINTER TO IPersistentRecipeHelper;
	_BVALID : BOOL;
END_VAR
END_FUNCTION_BLOCK

METHOD COMPARE : BOOL
END_METHOD

METHOD DELETE : BOOL
END_METHOD

METHOD LOAD : BOOL
END_METHOD

METHOD LOADFROM : BOOL
VAR_INPUT
	STNAME : REFERENCE TO STRING(255);
END_VAR
END_METHOD

METHOD READ : BOOL
END_METHOD

METHOD READNOSAVE : BOOL
END_METHOD

METHOD RELEASE : BOOL
END_METHOD

METHOD SAVE : BOOL
END_METHOD

METHOD SAVEAS : BOOL
VAR_INPUT
	STNAME : REFERENCE TO STRING(255);
END_VAR
END_METHOD

METHOD UPDATEFROMVALUES : BOOL
VAR_INPUT
	DESC : RecipeDescription;
END_VAR
END_METHOD

METHOD WRITE : BOOL
END_METHOD

METHOD INTINITIALIZE : BOOL
VAR_INPUT
	RECIPE : IRecipe;
	PRECIPEDEF : POINTER TO RecipeDefinition;
END_VAR
END_METHOD

METHOD INTINVALIDATE : BOOL
END_METHOD

METHOD PRVCHECKVALID : BOOL
END_METHOD

(* ---- RECIPESEM.pou ---- *)
FUNCTION_BLOCK RECIPESEM
VAR
	_HSEM : RTS_IEC_HANDLE;
END_VAR
END_FUNCTION_BLOCK

METHOD ENTER
END_METHOD

METHOD FB_EXIT : BOOL
VAR_INPUT
	BINCOPYCODE : BOOL;
END_VAR
END_METHOD

METHOD FB_INIT
VAR_INPUT
	BINITRETAINS : BOOL;
	BINCOPYCODE : BOOL;
END_VAR
END_METHOD

METHOD LEAVE
END_METHOD

(* ---- TL_RECIPEMANAGER.pou ---- *)
FUNCTION_BLOCK TL_RECIPEMANAGER
VAR
	M_TEXTLISTFILE : STRING(255);
	_STNAMESPACE : STRING;
END_VAR
END_FUNCTION_BLOCK

(* ---- TXTMANYFILESPERSISTANTRECIPEHELPER.pou ---- *)
FUNCTION_BLOCK TXTMANYFILESPERSISTANTRECIPEHELPER
VAR
	_STDEFNAME : STRING;
	_STNOVARNAMEFOUND : STRING(20) := 'NoVariableNameFound';
	_STSEPARATOR : STRING(2) := ':=';
	_STNEWLINE : STRING(2) := '$R$N';
	_STCOLUMNS : STRING(40) := '0|1';
	_STEXTENSION : STRING(16) := '.txtrecipe';
	_STPATH : STRING(512) := '';
	_LOADTYPE : PersistantLoadType := PersistantLoadType.LOAD_TYPE_NONE;
	_RECIPEMANAGER : IRecipeManager;
	_DATABUFFER : ARRAY [0..MAX_BUFFER_SIZE] OF BYTE;
	_CURRENTDATAPOSITION : INT;
	_BWRITEASUTF8 : BOOL := FALSE;
	_BREADASUTF8 : BOOL := FALSE;
	_UTF8HEADER : DWORD := 16#BFBBEF;
	_MTRSS : MembersToReduceStackSize;
	MAX_BUFFER_SIZE : INT := 2000;
	RECIPEDEFINITIONNAME : STRING;
END_VAR
END_FUNCTION_BLOCK

METHOD DELETERECIPE : BOOL
VAR_INPUT
	STNAME : STRING;
END_VAR
END_METHOD

METHOD GETFILEEXTENSION : STRING
END_METHOD

METHOD GETFILEPATH : STRING(512)
END_METHOD

METHOD LOADRECIPE : BOOL
VAR_INPUT
	DESC : REFERENCE TO RecipeDescription;
END_VAR
END_METHOD

METHOD LOADRECIPEFROM : BOOL
VAR_INPUT
	DESC : REFERENCE TO RecipeDescription;
	STFILE : REFERENCE TO STRING(255);
END_VAR
END_METHOD

METHOD SAVERECIPE : BOOL
VAR_INPUT
	DESC : REFERENCE TO RecipeDescription;
END_VAR
END_METHOD

METHOD SAVERECIPEAS : BOOL
VAR_INPUT
	DESC : REFERENCE TO RecipeDescription;
	STFILE : REFERENCE TO STRING(255);
END_VAR
END_METHOD

METHOD SETFILEPATH : BOOL
VAR_INPUT
	STPATH : STRING(512);
END_VAR
END_METHOD

METHOD SETRECIPEMANAGER
VAR_INPUT
	RECIPEMANAGER : IRecipeManager;
END_VAR
END_METHOD

METHOD PRVINITFILENAME : BOOL
VAR_INPUT
	STRECIPE : STRING;
END_VAR
END_METHOD

METHOD PRVSETLASTERROR : BOOL
VAR_INPUT
	DWERROR : DWORD;
END_VAR
END_METHOD

METHOD PRVSETLASTINFO : BOOL
VAR_INPUT
	EINFO : InfoValues;
END_VAR
END_METHOD

METHOD PRVCHECKVARNAME : BOOL
VAR_INPUT
	PVARDESC : POINTER TO RecipeVariableDescription;
	PSTNAME : POINTER TO STRING(256);
	BENDSWITH : BOOL;
END_VAR
END_METHOD

METHOD PRVFINDNAME : BOOL
VAR_INPUT
	PRECDESC : POINTER TO RecipeDescriptionData;
	PSTNAME : POINTER TO STRING(256);
	PNPOS : POINTER TO DINT;
	BNAME : BOOL;
	BENDSWITH : BOOL;
	ISEARCHSTARTPOS : DINT;
END_VAR
END_METHOD

METHOD PRVGENERATEINFOIF : BOOL
VAR_INPUT
	PRECDESC : POINTER TO RecipeDescriptionData;
END_VAR
END_METHOD

METHOD PRVREADDATAVALUE : BOOL
VAR_INPUT
	DATA : POINTER TO BYTE;
	VALUE : IEC_AnyType;
END_VAR
END_METHOD

METHOD PRVREADLINE : POINTER TO BYTE
VAR_INPUT
	PDATA : POINTER TO BYTE;
	PULSTART : POINTER TO DWORD;
	ULSIZE : DWORD;
END_VAR
END_METHOD

METHOD PRVRESETFLAGS : BOOL
VAR_INPUT
	PRECDESC : POINTER TO RecipeDescriptionData;
END_VAR
END_METHOD

METHOD PRVTRYTOFINDVARIABLENAMEPOS : DINT
VAR_INPUT
	DESC : REFERENCE TO RecipeDescription;
	PSTVALUE : POINTER TO STRING;
	STRDELIMS : STRING;
	DIPOSVARNAME : DINT;
	ISEARCHSTARTPOS : DINT;
END_VAR
END_METHOD

METHOD PRVGETCOMMENT : POINTER TO BYTE
VAR_INPUT
	PVARDESC : POINTER TO RecipeVariableDescription;
	PSTR : POINTER TO STRING(255);
	PILEN : POINTER TO INT;
END_VAR
END_METHOD

METHOD PRVGETMAX : POINTER TO BYTE
VAR_INPUT
	PVARDESC : POINTER TO RecipeVariableDescription;
	PSTR : POINTER TO STRING;
	PILEN : POINTER TO INT;
END_VAR
END_METHOD

METHOD PRVGETMIN : POINTER TO BYTE
VAR_INPUT
	PVARDESC : POINTER TO RecipeVariableDescription;
	PSTR : POINTER TO STRING;
	PILEN : POINTER TO INT;
END_VAR
END_METHOD

METHOD PRVGETNAME : POINTER TO BYTE
VAR_INPUT
	PVARDESC : POINTER TO RecipeVariableDescription;
	PILEN : POINTER TO INT;
END_VAR
END_METHOD

METHOD PRVGETTYPE : POINTER TO BYTE
VAR_INPUT
	VALUE : IEC_AnyType;
	PSTR : POINTER TO STRING(255);
	IBUFFERSIZE : INT;
	PILEN : POINTER TO INT;
END_VAR
END_METHOD

METHOD PRVGETVALUE : POINTER TO BYTE
VAR_INPUT
	VALUE : IEC_AnyType;
	PSTR : POINTER TO BYTE;
	IBUFFERSIZE : INT;
	PILEN : POINTER TO INT;
END_VAR
END_METHOD

METHOD PRVGETVARNAME : POINTER TO BYTE
VAR_INPUT
	PVARDESC : POINTER TO RecipeVariableDescription;
	PILEN : POINTER TO INT;
END_VAR
END_METHOD

METHOD PRVMEMCOPY : BOOL
VAR_INPUT
	PMEMDEST : POINTER TO BYTE;
	PMEMSOURCE : POINTER TO BYTE;
	ISIZE : INT;
END_VAR
END_METHOD

METHOD PRVSAVERECIPEBUFFERED : BOOL
VAR_INPUT
	DESC : REFERENCE TO RecipeDescription;
	DWHANDLE : SysFile.RTS_IEC_HANDLE;
END_VAR
END_METHOD

METHOD PRVWRITEDATAVALUE : BOOL
VAR_INPUT
	PVARDESC : POINTER TO RecipeVariableDescription;
	VALUE : IEC_AnyType;
	DWFILE : SysFile.RTS_IEC_HANDLE;
END_VAR
END_METHOD

METHOD PRVWRITEVALUE : BOOL
VAR_INPUT
	PDATA : POINTER TO BYTE;
	ISIZE : INT;
	DWFILE : SysFile.RTS_IEC_HANDLE;
END_VAR
END_METHOD

(* ---- VISU_FBCREATERECIPE.pou ---- *)
FUNCTION_BLOCK VISU_FBCREATERECIPE EXTENDS AbstractRecipeAndDefinitionNameCommand
END_FUNCTION_BLOCK

METHOD EXECUTEONRECIPEDEFINITIONANDRECIPENAME : DWORD
VAR_INPUT
	STRECIPEDEFINITIONNAME : STRING;
	STRECIPENAME : STRING;
END_VAR
END_METHOD

(* ---- VISU_FBDELETERECIPE.pou ---- *)
FUNCTION_BLOCK VISU_FBDELETERECIPE EXTENDS AbstractRecipeAndDefinitionNameCommand
END_FUNCTION_BLOCK

METHOD EXECUTEONRECIPEDEFINITIONANDRECIPENAME : DWORD
VAR_INPUT
	STRECIPEDEFINITIONNAME : STRING;
	STRECIPENAME : STRING;
END_VAR
END_METHOD

(* ---- VISU_FBDELETERECIPEFILE.pou ---- *)
FUNCTION_BLOCK VISU_FBDELETERECIPEFILE EXTENDS AbstractRecipeAndDefinitionNameCommand
END_FUNCTION_BLOCK

METHOD EXECUTEONRECIPEDEFINITIONANDRECIPENAME : DWORD
VAR_INPUT
	STRECIPEDEFINITIONNAME : STRING;
	STRECIPENAME : STRING;
END_VAR
END_METHOD

(* ---- VISU_FBFILEEXTENSIONANDPATH.pou ---- *)
FUNCTION_BLOCK VISU_FBFILEEXTENSIONANDPATH EXTENDS AbstractGeneralCommand
END_FUNCTION_BLOCK

METHOD EXECUTE : __XWORD
VAR_INPUT
	DWPARAM1 : __XWORD;
	DWPARAM2 : __XWORD;
END_VAR
END_METHOD

(* ---- VISU_FBLOADFROMANDWRITERECIPE.pou ---- *)
FUNCTION_BLOCK VISU_FBLOADFROMANDWRITERECIPE EXTENDS AbstractFileParamsCommand
END_FUNCTION_BLOCK

METHOD EXECUTEONFILEPARAMS : DWORD
VAR_INPUT
	STRECIPEDEF : STRING;
	STRECIPENAME : STRING;
	STFILE : STRING(255);
END_VAR
END_METHOD

(* ---- VISU_FBLOADFROMRECIPE.pou ---- *)
FUNCTION_BLOCK VISU_FBLOADFROMRECIPE EXTENDS AbstractFileParamsCommand
END_FUNCTION_BLOCK

METHOD EXECUTEONFILEPARAMS : DWORD
VAR_INPUT
	STRECIPEDEF : STRING;
	STRECIPENAME : STRING;
	STFILE : STRING(255);
END_VAR
END_METHOD

(* ---- VISU_FBLOADRECIPE.pou ---- *)
FUNCTION_BLOCK VISU_FBLOADRECIPE EXTENDS AbstractRecipeAndDefinitionNameCommand
END_FUNCTION_BLOCK

METHOD EXECUTEONRECIPEDEFINITIONANDRECIPENAME : DWORD
VAR_INPUT
	STRECIPEDEFINITIONNAME : STRING;
	STRECIPENAME : STRING;
END_VAR
END_METHOD

(* ---- VISU_FBREADANDSAVEASRECIPE.pou ---- *)
FUNCTION_BLOCK VISU_FBREADANDSAVEASRECIPE EXTENDS AbstractFileParamsCommand
VAR
	_XCHECKOVERWRITE : BOOL := TRUE;
	_MESSAGEBOXINFO : MessageBox_Struct;
	_MESSAGEBOXINFOBUSY : MessageBox_Struct;
	_FBOPENDIALOG : VU.FbOpenDialogExtended;
	_FBOPENBUSYDIALOG : VU.FbOpenDialogExtended;
	_ITFDIALOGCLOSEDLISTENER : VU.VisuElemBase.IDialogCloseListener := THIS^;
	_STRECIPEDEF : STRING;
	_STRECIPENAME : STRING;
	_STFILE : STRING(255);
	_XBUSY : BOOL;
END_VAR
END_FUNCTION_BLOCK

METHOD DIALOGCLOSED
VAR_INPUT
	ITFDIALOG : VU.VisuElemBase.IVisualisationDialog;
	PCLIENTDATA : POINTER TO VU.VisuElemBase.VisuStructClientData;
END_VAR
END_METHOD

METHOD EXECUTEONFILEPARAMS : DWORD
VAR_INPUT
	STRECIPEDEF : STRING;
	STRECIPENAME : STRING;
	STFILE : STRING(255);
END_VAR
END_METHOD

METHOD OPENBUSYDIALOG : BOOL
END_METHOD

METHOD OPENCHECKOVERWRITEDIALOG : BOOL
END_METHOD

(* ---- VISU_FBREADRECIPE.pou ---- *)
FUNCTION_BLOCK VISU_FBREADRECIPE EXTENDS AbstractRecipeAndDefinitionNameCommand
END_FUNCTION_BLOCK

METHOD EXECUTEONRECIPEDEFINITIONANDRECIPENAME : DWORD
VAR_INPUT
	STRECIPEDEFINITIONNAME : STRING;
	STRECIPENAME : STRING;
END_VAR
END_METHOD

(* ---- VISU_FBSAVEASRECIPE.pou ---- *)
FUNCTION_BLOCK VISU_FBSAVEASRECIPE EXTENDS Visu_FbReadAndSaveAsRecipe
END_FUNCTION_BLOCK

(* ---- VISU_FBSAVERECIPE.pou ---- *)
FUNCTION_BLOCK VISU_FBSAVERECIPE EXTENDS AbstractRecipeAndDefinitionNameCommand
END_FUNCTION_BLOCK

METHOD EXECUTEONRECIPEDEFINITIONANDRECIPENAME : DWORD
VAR_INPUT
	STRECIPEDEFINITIONNAME : STRING;
	STRECIPENAME : STRING;
END_VAR
END_METHOD

(* ---- VISU_FBSELECTRECIPE.pou ---- *)
FUNCTION_BLOCK VISU_FBSELECTRECIPE EXTENDS AbstractGeneralCommand
END_FUNCTION_BLOCK

METHOD EXECUTE : __XWORD
VAR_INPUT
	DWPARAM1 : __XWORD;
	DWPARAM2 : __XWORD;
END_VAR
END_METHOD

(* ---- VISU_FBSELECTRECIPEDEFINITION.pou ---- *)
FUNCTION_BLOCK VISU_FBSELECTRECIPEDEFINITION EXTENDS AbstractGeneralCommand
END_FUNCTION_BLOCK

METHOD EXECUTE : __XWORD
VAR_INPUT
	DWPARAM1 : __XWORD;
	DWPARAM2 : __XWORD;
END_VAR
END_METHOD

(* ---- VISU_FBWRITERECIPE.pou ---- *)
FUNCTION_BLOCK VISU_FBWRITERECIPE EXTENDS AbstractRecipeAndDefinitionNameCommand
END_FUNCTION_BLOCK

METHOD EXECUTEONRECIPEDEFINITIONANDRECIPENAME : DWORD
VAR_INPUT
	STRECIPEDEFINITIONNAME : STRING;
	STRECIPENAME : STRING;
END_VAR
END_METHOD

(* ---- VISU_RECIPECOMMANDS.pou ---- *)
FUNCTION_BLOCK VISU_RECIPECOMMANDS
VAR
	_CMDSELECTRECIPEDEFINITION : Visu_FbSelectRecipeDefinition;
	_CMDSELECTRECIPE : Visu_FbSelectRecipe;
	_CMDREADRECIPE : Visu_FbReadRecipe;
	_CMDWRITERECIPE : Visu_FbWriteRecipe;
	_CMDLOADRECIPE : Visu_FbLoadRecipe;
	_CMDSAVERECIPE : Visu_FbSaveRecipe;
	_CMDCREATERECIPE : Visu_FbCreateRecipe;
	_CMDDELETERECIPE : Visu_FbDeleteRecipe;
	_CMDRECIPELOADFROM : Visu_FbLoadFromRecipe;
	_CMDFILEEXTENSIONANDPATH : Visu_FbFileExtensionAndPath;
	_RECIPEMANAGER : IRecipeManager;
	_MEMORYFORCMDRECIPESAVEAS : POINTER TO BYTE;
END_VAR
END_FUNCTION_BLOCK

METHOD FB_EXIT : BOOL
VAR_INPUT
	BINCOPYCODE : BOOL;
END_VAR
END_METHOD

METHOD FB_INIT
VAR_INPUT
	BINITRETAINS : BOOL;
	BINCOPYCODE : BOOL;
	RECIPEMANAGER : IRecipeManager;
END_VAR
END_METHOD

METHOD REGISTERCOMMANDS : BOOL
VAR_INPUT
	COMMANDMANAGER : ICommandManager2;
END_VAR
END_METHOD

METHOD SETRECIPEMANAGER : DWORD
VAR_INPUT
	RECIPEMANAGER : IRecipeManager;
END_VAR
END_METHOD
